# EPICS autosave request: FOFBApp/Db/FOFBCtrl_settings.req
$(P)$(R)$(FOFB_CC)CCEnable-SP
$(P)$(R)$(FOFB_CC)TFSOverride-SP
$(P)$(R)$(FOFB_CC)BPMId-SP
$(P)$(R)$(FOFB_CC)TimeFrameLen-SP
$(P)$(R)$(FOFB_CC)MgtPowerdown-SP
$(P)$(R)$(FOFB_CC)MgtLoopback-SP
$(P)$(R)$(FOFB_CC)TimeFrameDly-SP
$(P)$(R)$(FOFB_CC)GoldenOrbX-SP
$(P)$(R)$(FOFB_CC)GoldenOrbY-SP
$(P)$(R)$(FOFB_CC)CustFeature-SP
$(P)$(R)$(FOFB_CC)RxPolarity-SP
$(P)$(R)$(FOFB_CC)PayloadSel-SP
$(P)$(R)$(FOFB_CC)DataSel-SP
$(P)$(R)$(FOFB_CC)TOARdEn-SP
$(P)$(R)$(FOFB_CC)RCBRdEn-SP
